// TIA Portal project "Girello_automatico2" (V15.1)

(* hardware
DEVICE "S7-1200 station_1"  S7-1200 Station
   slot 0: "Telaio di montaggio_0"  S7-1200 Rack  Rack  V1.0
   slot 1: "PLC_1"  CPU 1214C DC/DC/DC  6ES7 214-1AG40-0XB0  V4.2
*)

// ===== PLC "PLC_1"  CPU 1214C DC/DC/DC =====

VAR_GLOBAL   // PLC tag table "Tabella delle variabili standard"
   "P1" AT %I0.0 : Bool;
   "P2" AT %I0.1 : Bool;
   "PG" AT %I0.2 : Bool;
   "PX" AT %I0.3 : Bool;
   "FCS" AT %I0.4 : Bool;
   "FCD" AT %I0.5 : Bool;
   "M1" AT %Q0.0 : Bool;
   "M2" AT %Q0.1 : Bool;
   "MG" AT %Q0.2 : Bool;
   "S" AT %Q0.3 : Bool;
   "D" AT %Q0.4 : Bool;
END_VAR

DATA_BLOCK "variabili_stato1"   // DB1
{ S7_Optimized_Access := 'TRUE' }
VERSION : 0.1
   VAR RETAIN
      home : Bool := true;
      muovi1 : Bool;
      wait : Bool;
      muovi2 : Bool;
   END_VAR
BEGIN
END_DATA_BLOCK

DATA_BLOCK "variabili_statoG"   // DB2
{ S7_Optimized_Access := 'TRUE' }
VERSION : 0.1
   VAR RETAIN
      home : Bool := true;
      muovi : Bool;
      ruotaS : Bool;
      ruotaD : Bool;
      wait1 : Bool;
      wait2 : Bool;
   END_VAR
BEGIN
END_DATA_BLOCK

DATA_BLOCK "variabili_stato2"   // DB3
{ S7_Optimized_Access := 'TRUE' }
VERSION : 0.1
   VAR RETAIN
      home : Bool := true;
      muovi : Bool;
      wait : Bool;
   END_VAR
BEGIN
END_DATA_BLOCK

ORGANIZATION_BLOCK "nastro1"   // OB1, LAD, ProgramCycle
TITLE = "Main Program Sweep (Cycle)"
{ S7_Optimized_Access := 'TRUE' }
VERSION : 0.1
   VAR_INPUT
      Initial_Call : Bool;   // Initial call of this OB
      Remanence : Bool;   // =True, if remanent data are available
   END_VAR
BEGIN

REGION Network 1
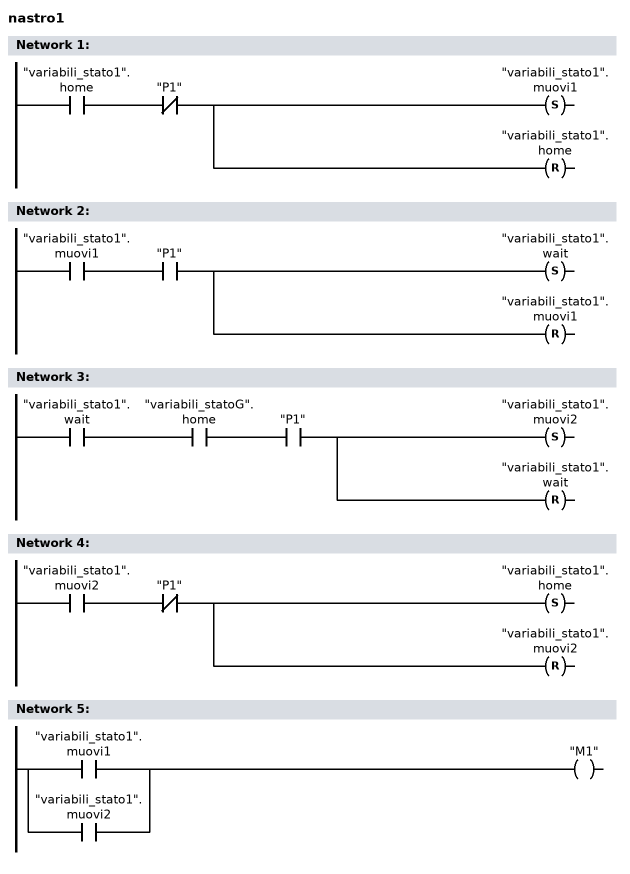
   RUNG wire#powerrail
      Contact( "variabili_stato1".home )
      I_Contact( "P1" )
      wire#w1
      S_Coil( "variabili_stato1".muovi1 )
   END_RUNG
   RUNG wire#w1
      R_Coil( "variabili_stato1".home )
   END_RUNG
   // the same network as SCL:
   IF "variabili_stato1".home AND NOT "P1" THEN
       "variabili_stato1".muovi1 := TRUE;
       "variabili_stato1".home := FALSE;
   END_IF;
END_REGION

REGION Network 2
   RUNG wire#powerrail
      Contact( "variabili_stato1".muovi1 )
      Contact( "P1" )
      wire#w1
      S_Coil( "variabili_stato1".wait )
   END_RUNG
   RUNG wire#w1
      R_Coil( "variabili_stato1".muovi1 )
   END_RUNG
   // the same network as SCL:
   IF "variabili_stato1".muovi1 AND "P1" THEN
       "variabili_stato1".wait := TRUE;
       "variabili_stato1".muovi1 := FALSE;
   END_IF;
END_REGION

REGION Network 3
   RUNG wire#powerrail
      Contact( "variabili_stato1".wait )
      Contact( "variabili_statoG".home )
      Contact( "P1" )
      wire#w1
      S_Coil( "variabili_stato1".muovi2 )
   END_RUNG
   RUNG wire#w1
      R_Coil( "variabili_stato1".wait )
   END_RUNG
   // the same network as SCL:
   IF "variabili_stato1".wait AND "variabili_statoG".home AND "P1" THEN
       "variabili_stato1".muovi2 := TRUE;
       "variabili_stato1".wait := FALSE;
   END_IF;
END_REGION

REGION Network 4
   RUNG wire#powerrail
      Contact( "variabili_stato1".muovi2 )
      I_Contact( "P1" )
      wire#w1
      S_Coil( "variabili_stato1".home )
   END_RUNG
   RUNG wire#w1
      R_Coil( "variabili_stato1".muovi2 )
   END_RUNG
   // the same network as SCL:
   IF "variabili_stato1".muovi2 AND NOT "P1" THEN
       "variabili_stato1".home := TRUE;
       "variabili_stato1".muovi2 := FALSE;
   END_IF;
END_REGION

REGION Network 5
   RUNG wire#powerrail
      Contact( "variabili_stato1".muovi1 )
      wire#w1
      Coil( "M1" )
   END_RUNG
   RUNG wire#powerrail
      Contact( "variabili_stato1".muovi2 )
   END_RUNG wire#w1
   // the same network as SCL:
   "M1" := "variabili_stato1".muovi1 OR "variabili_stato1".muovi2;
END_REGION
END_ORGANIZATION_BLOCK

ORGANIZATION_BLOCK "girello"   // OB123, LAD, ProgramCycle
TITLE = "Main Program Sweep (Cycle)"
{ S7_Optimized_Access := 'TRUE' }
VERSION : 0.1
   VAR_INPUT
      Initial_Call : Bool;   // Initial call of this OB
      Remanence : Bool;   // =True, if remanent data are available
   END_VAR
BEGIN

REGION Network 1
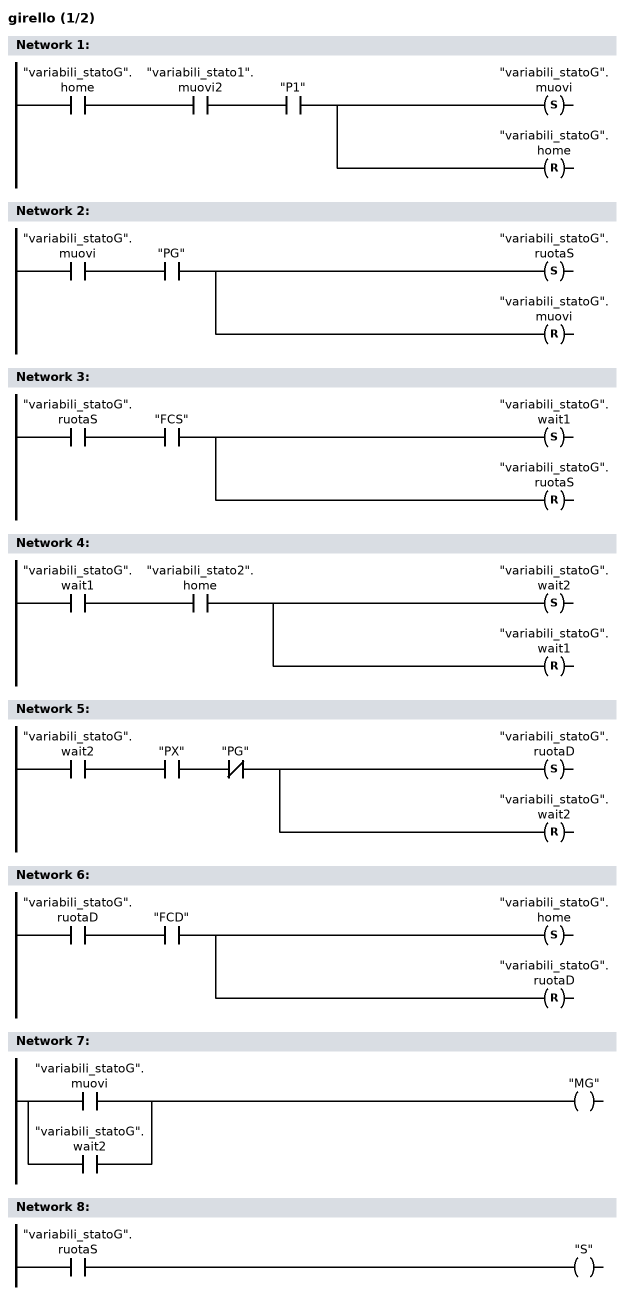
   RUNG wire#powerrail
      Contact( "variabili_statoG".home )
      Contact( "variabili_stato1".muovi2 )
      Contact( "P1" )
      wire#w1
      S_Coil( "variabili_statoG".muovi )
   END_RUNG
   RUNG wire#w1
      R_Coil( "variabili_statoG".home )
   END_RUNG
   // the same network as SCL:
   IF "variabili_statoG".home AND "variabili_stato1".muovi2 AND "P1" THEN
       "variabili_statoG".muovi := TRUE;
       "variabili_statoG".home := FALSE;
   END_IF;
END_REGION

REGION Network 2
   RUNG wire#powerrail
      Contact( "variabili_statoG".muovi )
      Contact( "PG" )
      wire#w1
      S_Coil( "variabili_statoG".ruotaS )
   END_RUNG
   RUNG wire#w1
      R_Coil( "variabili_statoG".muovi )
   END_RUNG
   // the same network as SCL:
   IF "variabili_statoG".muovi AND "PG" THEN
       "variabili_statoG".ruotaS := TRUE;
       "variabili_statoG".muovi := FALSE;
   END_IF;
END_REGION

REGION Network 3
   RUNG wire#powerrail
      Contact( "variabili_statoG".ruotaS )
      Contact( "FCS" )
      wire#w1
      S_Coil( "variabili_statoG".wait1 )
   END_RUNG
   RUNG wire#w1
      R_Coil( "variabili_statoG".ruotaS )
   END_RUNG
   // the same network as SCL:
   IF "variabili_statoG".ruotaS AND "FCS" THEN
       "variabili_statoG".wait1 := TRUE;
       "variabili_statoG".ruotaS := FALSE;
   END_IF;
END_REGION

REGION Network 4
   RUNG wire#powerrail
      Contact( "variabili_statoG".wait1 )
      Contact( "variabili_stato2".home )
      wire#w1
      S_Coil( "variabili_statoG".wait2 )
   END_RUNG
   RUNG wire#w1
      R_Coil( "variabili_statoG".wait1 )
   END_RUNG
   // the same network as SCL:
   IF "variabili_statoG".wait1 AND "variabili_stato2".home THEN
       "variabili_statoG".wait2 := TRUE;
       "variabili_statoG".wait1 := FALSE;
   END_IF;
END_REGION

REGION Network 5
   RUNG wire#powerrail
      Contact( "variabili_statoG".wait2 )
      Contact( "PX" )
      I_Contact( "PG" )
      wire#w1
      S_Coil( "variabili_statoG".ruotaD )
   END_RUNG
   RUNG wire#w1
      R_Coil( "variabili_statoG".wait2 )
   END_RUNG
   // the same network as SCL:
   IF "variabili_statoG".wait2 AND "PX" AND NOT "PG" THEN
       "variabili_statoG".ruotaD := TRUE;
       "variabili_statoG".wait2 := FALSE;
   END_IF;
END_REGION

REGION Network 6
   RUNG wire#powerrail
      Contact( "variabili_statoG".ruotaD )
      Contact( "FCD" )
      wire#w1
      S_Coil( "variabili_statoG".home )
   END_RUNG
   RUNG wire#w1
      R_Coil( "variabili_statoG".ruotaD )
   END_RUNG
   // the same network as SCL:
   IF "variabili_statoG".ruotaD AND "FCD" THEN
       "variabili_statoG".home := TRUE;
       "variabili_statoG".ruotaD := FALSE;
   END_IF;
END_REGION

REGION Network 7
   RUNG wire#powerrail
      Contact( "variabili_statoG".muovi )
      wire#w1
      Coil( "MG" )
   END_RUNG
   RUNG wire#powerrail
      Contact( "variabili_statoG".wait2 )
   END_RUNG wire#w1
   // the same network as SCL:
   "MG" := "variabili_statoG".muovi OR "variabili_statoG".wait2;
END_REGION

REGION Network 8
   RUNG wire#powerrail
      Contact( "variabili_statoG".ruotaS )
      Coil( "S" )
   END_RUNG
   // the same network as SCL:
   "S" := "variabili_statoG".ruotaS;
END_REGION

REGION Network 9
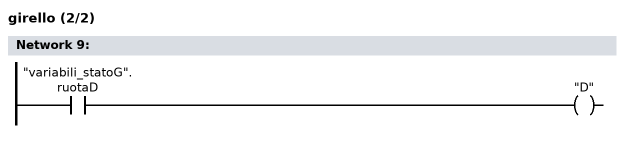
   RUNG wire#powerrail
      Contact( "variabili_statoG".ruotaD )
      Coil( "D" )
   END_RUNG
   // the same network as SCL:
   "D" := "variabili_statoG".ruotaD;
END_REGION
END_ORGANIZATION_BLOCK

ORGANIZATION_BLOCK "nastro2"   // OB124, LAD, ProgramCycle
TITLE = "Main Program Sweep (Cycle)"
{ S7_Optimized_Access := 'TRUE' }
VERSION : 0.1
   VAR_INPUT
      Initial_Call : Bool;   // Initial call of this OB
      Remanence : Bool;   // =True, if remanent data are available
   END_VAR
BEGIN

REGION Network 1
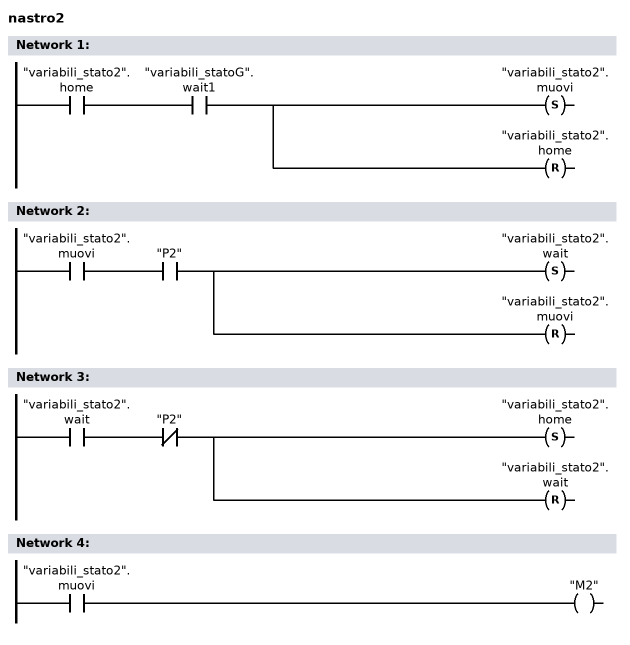
   RUNG wire#powerrail
      Contact( "variabili_stato2".home )
      Contact( "variabili_statoG".wait1 )
      wire#w1
      S_Coil( "variabili_stato2".muovi )
   END_RUNG
   RUNG wire#w1
      R_Coil( "variabili_stato2".home )
   END_RUNG
   // the same network as SCL:
   IF "variabili_stato2".home AND "variabili_statoG".wait1 THEN
       "variabili_stato2".muovi := TRUE;
       "variabili_stato2".home := FALSE;
   END_IF;
END_REGION

REGION Network 2
   RUNG wire#powerrail
      Contact( "variabili_stato2".muovi )
      Contact( "P2" )
      wire#w1
      S_Coil( "variabili_stato2".wait )
   END_RUNG
   RUNG wire#w1
      R_Coil( "variabili_stato2".muovi )
   END_RUNG
   // the same network as SCL:
   IF "variabili_stato2".muovi AND "P2" THEN
       "variabili_stato2".wait := TRUE;
       "variabili_stato2".muovi := FALSE;
   END_IF;
END_REGION

REGION Network 3
   RUNG wire#powerrail
      Contact( "variabili_stato2".wait )
      I_Contact( "P2" )
      wire#w1
      S_Coil( "variabili_stato2".home )
   END_RUNG
   RUNG wire#w1
      R_Coil( "variabili_stato2".wait )
   END_RUNG
   // the same network as SCL:
   IF "variabili_stato2".wait AND NOT "P2" THEN
       "variabili_stato2".home := TRUE;
       "variabili_stato2".wait := FALSE;
   END_IF;
END_REGION

REGION Network 4
   RUNG wire#powerrail
      Contact( "variabili_stato2".muovi )
      Coil( "M2" )
   END_RUNG
   // the same network as SCL:
   "M2" := "variabili_stato2".muovi;
END_REGION
END_ORGANIZATION_BLOCK